TYPE
    ComRobOut :
    STRUCT
        {attribute addProperty Name "<#AutoMode Aktiv#>"}
        ModeAuto        : BOOL;
        stopRun         : BOOL;
        reset           : BOOL;
        contactReady    : BOOL;
        contactPunched  : BOOL;
        homePosReq      : BOOL;
        tableInPos      : BOOL;
        HighPowerOn     : BOOL;
        PalletPickIndex : INT := 0;
        HighPowerOff    : BOOL;
        RowDone         : BOOL;
        //auf HMI: 
        //            - Toggle vor eindruecken der Kontakte
        //              - Hoehe einstellbar
        ContactHeight        : INT;
        WaitBeforeContacting : BOOL;
        {attribute addProperty Name "<#Foto Done#>"}
        FotoDone  : BOOL;
        Locations : Locations;
    END_STRUCT
END_TYPE

(* stored: Version 1.1.0.1, ProductVersion 3.1.4024.12
   DUT ComRobOut: Id {85dca0dc-6b78-0813-3849-7013a0aeabff} *)
